(* IEC 61131-3 sources: TcTidier/tests/integration/workspace-template, 2 files *)

(* ---- document-format.expected.st ---- *)
PROGRAM DocumentFormatFixture
VAR
    flag    : BOOL;
    counter : INT;
END_VAR
IF flag THEN
    counter := counter+1;
END_IF

(* ---- document-format.st ---- *)
PROGRAM DocumentFormatFixture
VAR
flag:BOOL;
counter:INT;
END_VAR
IF flag THEN counter:=counter+1; END_IF
